PROGRAM TEST_BUFFERING
VAR
	fbRunAxis : POINTER TO RunAxis := ADR(GVL.axisControls[1]);
	
	
	ptCommand1 : POINTER TO ParameterSet := ADR(GVL.commandBlocks[8]);
	ptCommand2 : POINTER TO ParameterSet := ADR(GVL.commandBlocks[9]);
	ptCommand3 : POINTER TO ParameterSet := ADR(GVL.commandBlocks[10]);
	
	state : INT;
	
	bAction : bool;
	bDone1 : BOOL;
	bDone2 : BOOL;
	bDone3 : BOOL;
END_VAR

fbRunAxis^();

//master move with serveral buffers
//if bAction set to off when executing second command?
//return;

IF NOT bDone1 THEN
	bDone1 := fbRunAxis^.ExecuteParameterBuffer(ptBlock:=ptCommand1,
		bufferIndex:=1);
END_IF
IF NOT bDone2 AND (fbRunAxis^.PositionFeedback >= 250)  THEN
	bDone2 := fbRunAxis^.ExecuteParameterBuffer(ptBlock:=ptCommand2,
		bufferIndex:=2);
END_IF
IF NOT bDone3  AND (fbRunAxis^.PositionFeedback >=350)  THEN
	bDone3 := fbRunAxis^.ExecuteParameterBuffer(ptBlock:=ptCommand3,
		bufferIndex:=3);
END_IF

END_PROGRAM

(* stored: Version 1.1.0.1, ProductVersion 3.1.4022.10
   POU TEST_BUFFERING: Id {b3f04993-5876-444e-93e2-12f05fde09bf}, SpecialFunc None *)
